// TIA Portal V20 export
DATA_BLOCK "Axis_1"   // DB2
   // technology object, version 
BEGIN
END_DATA_BLOCK
